// TIA Portal V20 export
DATA_BLOCK "Volumeflow_outlet_DB"   // DB4
// stored: InstanceOfName Volumeflow, InstanceOfType FB
"Volumeflow"
   // VAR_INPUT
   //    Enable : Bool;
   //    Release_Spd : Int;
   //    T_Release : Real;
   //    Raw_Scale { ExternalAccessible := 'False'; ExternalVisible := 'False'; ExternalWritable := 'False'} : "ScaVal_Raw";
   // END_VAR
   // VAR_OUTPUT
   //    Liter : Real;
   //    Liters_Raw : Int;
   // END_VAR
   // VAR
   //    pi : Real;
   //    r : Real;
   // END_VAR
BEGIN
END_DATA_BLOCK
